{attribute 'linkalways'} 
{attribute 'no_explicit_call' := 'This FB is a CLASS and must be accessed using methods or properties'}
{attribute 'enable_dynamic_creation'}
FUNCTION_BLOCK FINAL MOD_LWORD EXTENDS Node
VAR
	in1 : _LWORD(0);
	in2 : _LWORD(0);
	out : _LWORD(0);
END_VAR

METHOD PUBLIC Clone : I_Node
VAR
	pNode : POINTER TO MOD_LWORD;
END_VAR
pNode := __NEW(MOD_LWORD);
Clone := pNode^;
END_METHOD

METHOD FB_init : BOOL
VAR_INPUT
	bInitRetains : BOOL; // if TRUE, the retain variables are initialized (warm start / cold start)
	bInCopyCode : BOOL;  // if TRUE, the instance afterwards gets moved into the copy code (online change)
END_VAR
AddInput('in1',THIS^.in1);
AddInput('in2',THIS^.in2);
AddOutput('out', THIS^.out);
END_METHOD

METHOD PROTECTED OnExecute
VAR
END_VAR
out.Value := in1.Value MOD in2.Value;
END_METHOD

END_FUNCTION_BLOCK

(* stored: Version 1.1.0.1, ProductVersion 3.1.4024.15
   POU MOD_LWORD: Id {f68ff752-3883-4638-9c0f-3485ee3821fd}, SpecialFunc None
   Folder Constructor: Id {75674312-80b7-4e83-9697-0f8d7c73532a}
   Method Clone: Id {b00df151-2c56-4b52-9b63-ce1ab972c770}
   Method FB_init: Id {4113720a-5109-4ef3-898d-2e324d0ae58f}
   Method OnExecute: Id {dbb7feca-ff11-4757-94cb-151e0f9f816a} *)
